// TIA Portal V20 export
FUNCTION_BLOCK "LER_E5CC"   // FB23, LAD
// stored: Access Published, MemoryReserve 100, SetENOAutomatically false
   VAR_INPUT
      enable : Bool;
      clock : Bool;
      unitNo : Int;
      save : Bool;
      Reset : Bool;
      AllHeaterRun : Bool;
      AllHeaterStop : Bool;
      AllHeaterAutoTuneRun : Bool;
      AllHeaterAutoTuneStop : Bool;
      HeaterCommands : "LER_typeE5CCCommands";
      HeaterConfiguration : "LER_typeE5CCConfiguration";
   END_VAR
   VAR_OUTPUT
      HeaterMonitoring : "LER_typeE5CCMonitoring";
   END_VAR
   VAR_IN_OUT
      CurrentUnit : Int;
      MBMasterBuffer : "LER_typeHeaterConfiguration_MB_Master";
   END_VAR
   VAR
      statHeaterRun : Bool;
      statHeaterStop : Bool;
      statHeaterAutoTuneRun : Bool;
      statHeaterAutoTuneStop : Bool;
      statReadStep : Int;
      statReadReq : Array[0..9] of Bool;
      statWriteReq : Array[0..9] of Bool;
      statPulse : Array[0..19] of Bool;
      statTimer { S7_SetPoint := 'True'} : Array[0..9] of TON_TIME;
      statReadTempPV : Real;
      statReadStatus : DWord;
      statTempSP : Real;
      statAlarmValue1 : Real;
      statAlarmValue1_UpperLimit : Real;
      statAlarmValue1_LowerLimit : Real;
      statAlarmValue2 : Real;
      statAlarmValue2_UpperLimit : Real;
      statAlarmValue2_LowerLimit : Real;
      statReadStatus_Bool : Array[0..31] of Bool;
      statHeater_PV_Buf : Real;
      statUpperComplete_Temp : Real;
      statLowerComplete_Temp : Real;
   END_VAR
   VAR_TEMP
      tempErr : Word;
   END_VAR
   VAR CONSTANT
      Addr_TempPV : UDInt := 40001;
      Addr_Status : UDInt := 40003;
      Addr_TempSP : UDInt := 40263;
      Addr_AlarmValue1 : UDInt := 40265;
      Addr_AlarmValue1_UpperLimit : UDInt := 40267;
      Addr_AlarmValue1_LowerLimit : UDInt := 40269;
      Addr_AlarmValue2 : UDInt := 40271;
      Addr_AlarmValue2_UpperLimit : UDInt := 40273;
      Addr_AlarmValue2_LowerLimit : UDInt := 40275;
      CMD_Run : DWord := 16#01000000;
      CMD_Stop : DWord := 16#01010000;
      CMD_AutoTune_Run : DWord := 16#03020000;
      CMD_AutoTune_Stop : DWord := 16#03000000;
      Mode_Read : Int := 0;
      Mode_Write : Int := 1;
      Read_Time : Time := T#1000MS;
      STATUS_NO_ERROR_OCCURRED : DWord;   // No error occurred.
      ERR_HEATER_CURRENT_VALUE_EXCEEDED_CT1 : DWord := 16#1;
      ERR_HEATER_CURRENT_VALUE_HOLD_CT1 : DWord := 16#2;
      ERR_AD_CONVERTER_ABNORMALITY : DWord := 16#4;
      ERR_HS_SSR_FAULT_ALERT_CT1 : DWord := 16#8;
      ERR_RSP_INPUT_ABNORMALITIES : DWord := 16#10;
      ERR_MORE_THAN_INPUT : DWord := 16#40;
      ERR_POTENTIOMETER_INPUT_ABNORMAL : DWord := 16#80;
      ERR_CONTROL_OUTPUT_HEATED_OPEN_OUTPUT : DWord := 16#100;
      ERR_CONTROL_OUTPUT_COOL_CLOSE_OUTPUT : DWord := 16#200;
      ERR_HEATER_OPEN_CIRCUIT_HB_ALARM_CT1 : DWord := 16#400;
      ERR_HEATER_OPEN_CIRCUIT_HB_ALARM_CT2 : DWord := 16#800;
      ERR_ALERT_1 : DWord := 16#1000;
      ERR_ALERT_2 : DWord := 16#2000;
      ERR_ALERT_3 : DWord := 16#4000;
      ERR_PROGRAM_END_OUTPUT : DWord := 16#8000;
      ERR_EVENT_INPUT_1 : DWord := 16#10000;
      ERR_EVENT_INPUT_2 : DWord := 16#20000;
      ERR_EVENT_INPUT_3 : DWord := 16#40000;
      ERR_EVENT_INPUT_4 : DWord := 16#80000;
      ERR_WRITE_MODE : DWord := 16#100000;
      ERR_NON_VOLATILE_MEMORY : DWord := 16#200000;
      ERR_SETTING_AREA : DWord := 16#400000;
      ERR_AT_RUN_STOP : DWord := 16#800000;
      ERR_RUN_STOP : DWord := 16#1000000;
      ERR_COMMUNICATION_WRITE : DWord := 16#2000000;
      ERR_AUTO_MANUAL : DWord := 16#4000000;
      ERR_PROGRAM_START : DWord := 16#8000000;
      ERR_HEATER_CURRENT_VALUE_EXCEEDED_CT2 : DWord := 16#10000000;
      ERR_HEATER_CURRENT_VALUE_HOLD_CT2 : DWord := 16#20000000;
      ERR_HS_SSR_FAILURE_ALARM_CT2 : DWord := 16#80000000;
   END_VAR
   // // statReadStatus_Bool[0] : Heater Current Value Exceeded (CT1)
   // // statReadStatus_Bool[1] : Heater Current Value Hold (CT1)
   // // statReadStatus_Bool[2] : AD converter abnormality
   // // statReadStatus_Bool[3] : HS (SSR Fault) Alert (CT1)
   // // statReadStatus_Bool[4] : RSP input abnormalities
   // // statReadStatus_Bool[6] : More than input
   // // statReadStatus_Bool[7] : Potenshometer input abnormal
   // // statReadStatus_Bool[8] : Control Output (Heated)/Open Output
   // // statReadStatus_Bool[9] : Control Output (Cool)/Close Output
   // // statReadStatus_Bool[10] : Heater Open Circuit (HB) Alarm (CT1)
   // // statReadStatus_Bool[11] : Heater Open Circuit (HB) Alarm (CT2)
   // // statReadStatus_Bool[12] : Alert 1
   // // statReadStatus_Bool[13] : Alert 2
   // // statReadStatus_Bool[14] : Alert 3
   // // statReadStatus_Bool[15] : Program END Output
   // // statReadStatus_Bool[16] : Event Input 1
   // // statReadStatus_Bool[17] : Event Input 2
   // // statReadStatus_Bool[18] : Event Input 3
   // // statReadStatus_Bool[19] : Event Input 4
   // // statReadStatus_Bool[20] : Write Mode
   // // statReadStatus_Bool[21] : Non-volatile Memory
   // // statReadStatus_Bool[22] : Setting Area
   // // statReadStatus_Bool[23] : AT Run/Stop
   // // statReadStatus_Bool[24] : RUN/STOP
   // // statReadStatus_Bool[25] : Communication Write
   // // statReadStatus_Bool[26] : Auto/Manual
   // // statReadStatus_Bool[27] : Program START
   // // statReadStatus_Bool[28] : Heater Current Value Exceeded (CT2)
   // // statReadStatus_Bool[29] : Heater Current Value Hold (CT2)
   // // statReadStatus_Bool[31] : HS (SSR Failure) Alarm (CT2)
   VAR_TEMP   // added for the SCL form of the ladder/FBD networks
      _w1 : Bool;
      _w2 : Bool;
   END_VAR
BEGIN

REGION Network 1 (SCL): ###### Input Mapping ######
   //Input Mapping
   #statHeaterRun := #AllHeaterRun OR #HeaterCommands.Heater_Run;
   #statHeaterStop := #AllHeaterStop OR #HeaterCommands.Heater_Stop;
   #statHeaterAutoTuneRun := #AllHeaterAutoTuneRun OR #HeaterCommands.AutoTune_Run;
   #statHeaterAutoTuneStop := #AllHeaterAutoTuneStop OR #HeaterCommands.AutoTune_Stop;

   //Read Step Initialization
   IF #statReadStep = 0 THEN
       #statReadStep := 1;
   ELSIF #statReadStep > 2 THEN
       #statReadStep := 1;
   END_IF;
END_REGION

REGION Network 2: Read Temp PV + Status Command
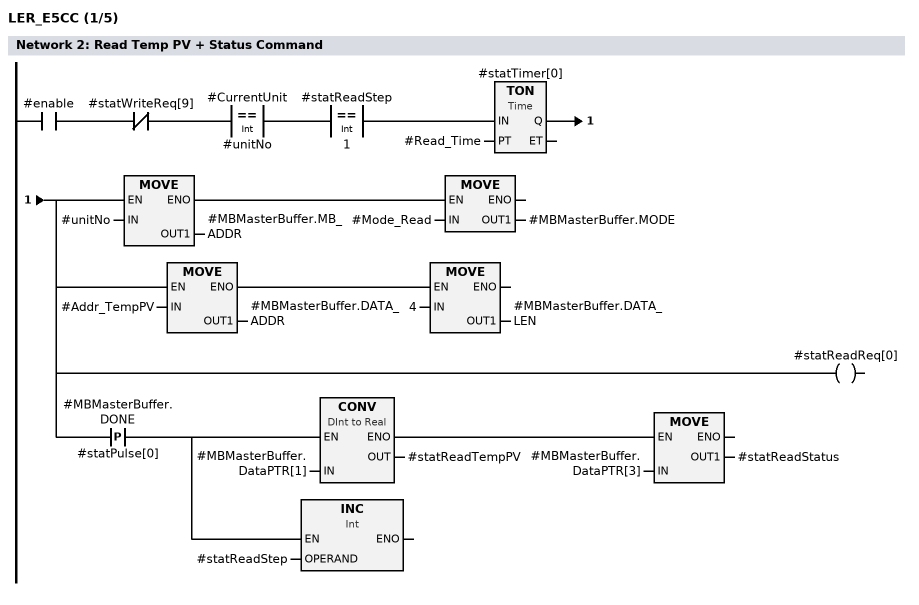
   RUNG wire#powerrail
      Contact( #enable )
      I_Contact( #statWriteReq[9] )
      { S7_Templates := "SrcType := Int" } EQ_Contact(in1 := #CurrentUnit, in2 := #unitNo)
      { S7_Templates := "SrcType := Int" } EQ_Contact(in1 := #statReadStep, in2 := 1)
      { S7_Templates := "time_type := Time" } #statTimer[0].TON(pt := #Read_Time, et =>)
      wire#w1
      Move(in := #unitNo, out1 => #MBMasterBuffer.MB_ADDR)
      Move(in := #Mode_Read, out1 => #MBMasterBuffer.MODE)
   END_RUNG
   RUNG wire#w1
      Move(in := #Addr_TempPV, out1 => #MBMasterBuffer.DATA_ADDR)
      Move(in := 4, out1 => #MBMasterBuffer.DATA_LEN)
   END_RUNG
   RUNG wire#w1
      Coil( #statReadReq[0] )
   END_RUNG
   RUNG wire#w1
      P_Contact(operand := #MBMasterBuffer.DONE, bit := #statPulse[0])
      wire#w2
      { S7_Templates := "[SrcType := DInt, DestType := Real]" } Convert(in := #MBMasterBuffer.DataPTR[1], out => #statReadTempPV)
      Move(in := #MBMasterBuffer.DataPTR[3], out1 => #statReadStatus)
   END_RUNG
   RUNG wire#w2
      { S7_Templates := "DestType := Int" } Inc( #statReadStep )
   END_RUNG
   // the same network as SCL:
   #statTimer[0].TON(IN := #enable AND NOT #statWriteReq[9] AND (#CurrentUnit = #unitNo) AND (#statReadStep = 1),
                     PT := #Read_Time);
   IF #statTimer[0].Q THEN
       #MBMasterBuffer.MB_ADDR := #unitNo;
       #MBMasterBuffer.MODE := #Mode_Read;
       #MBMasterBuffer.DATA_ADDR := #Addr_TempPV;
       #MBMasterBuffer.DATA_LEN := 4;
   END_IF;
   #statReadReq[0] := #statTimer[0].Q;
   #_w1 := #statTimer[0].Q AND #MBMasterBuffer.DONE AND NOT #statPulse[0];   // rising edge of #MBMasterBuffer.DONE
   #statPulse[0] := #MBMasterBuffer.DONE;
   IF #_w1 THEN
       #statReadTempPV := DINT_TO_REAL(#MBMasterBuffer.DataPTR[1]);
       #statReadStatus := #MBMasterBuffer.DataPTR[3];
       #statReadStep := #statReadStep + 1;
   END_IF;
END_REGION

REGION Network 3: Read TempSP + AlarmValue1 ~ AlarmValue2_LowerLimit Commad
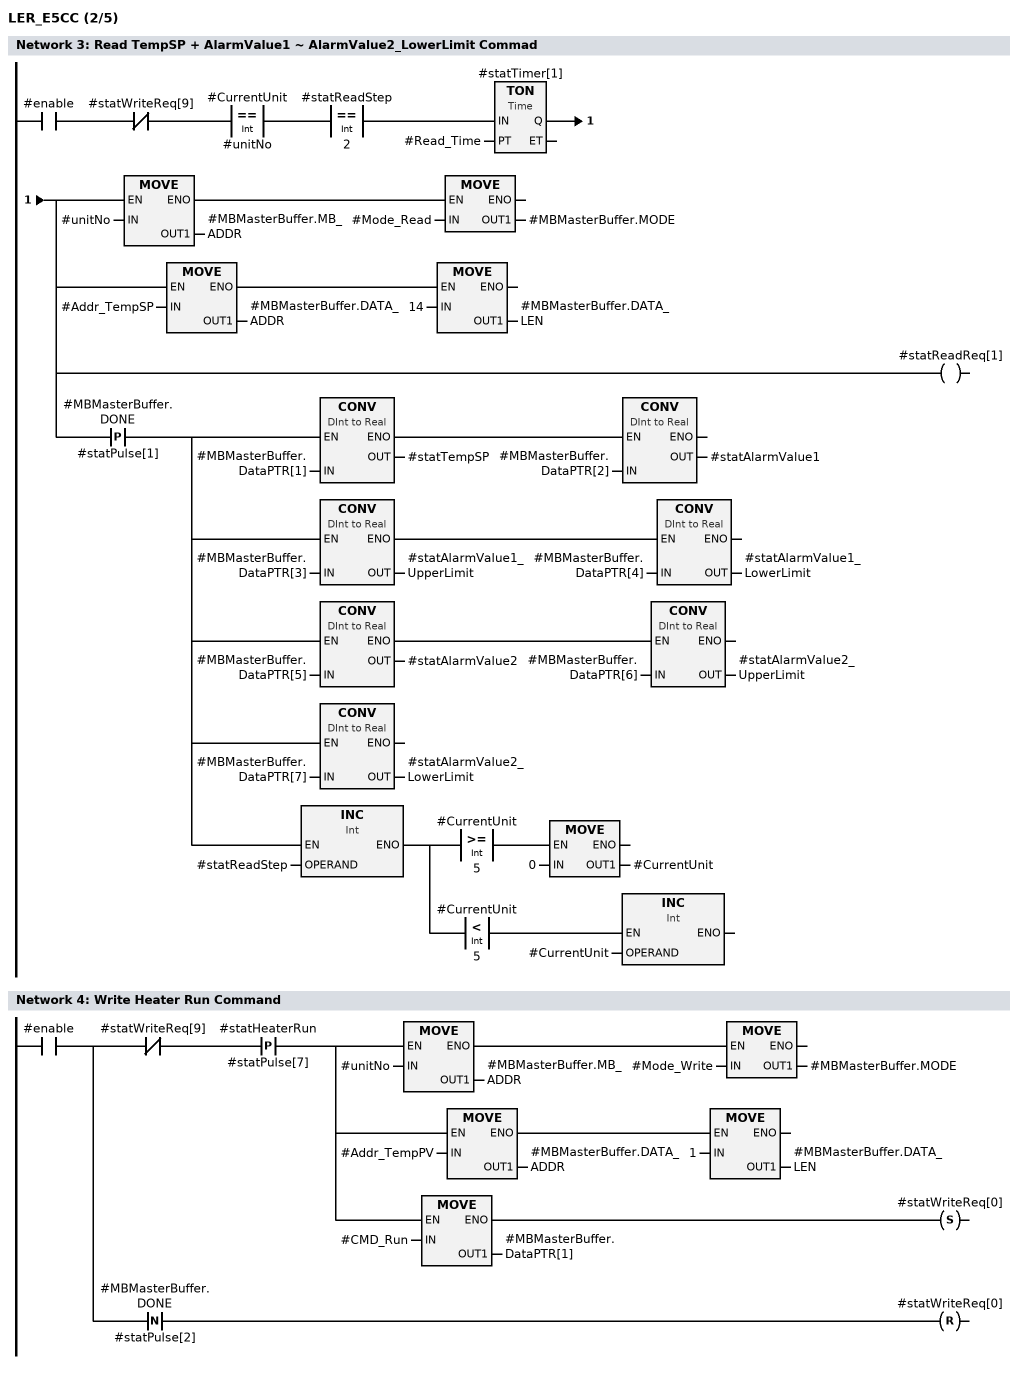
   RUNG wire#powerrail
      Contact( #enable )
      I_Contact( #statWriteReq[9] )
      { S7_Templates := "SrcType := Int" } EQ_Contact(in1 := #CurrentUnit, in2 := #unitNo)
      { S7_Templates := "SrcType := Int" } EQ_Contact(in1 := #statReadStep, in2 := 2)
      { S7_Templates := "time_type := Time" } #statTimer[1].TON(pt := #Read_Time, et =>)
      wire#w1
      Move(in := #unitNo, out1 => #MBMasterBuffer.MB_ADDR)
      Move(in := #Mode_Read, out1 => #MBMasterBuffer.MODE)
   END_RUNG
   RUNG wire#w1
      Move(in := #Addr_TempSP, out1 => #MBMasterBuffer.DATA_ADDR)
      Move(in := 14, out1 => #MBMasterBuffer.DATA_LEN)
   END_RUNG
   RUNG wire#w1
      Coil( #statReadReq[1] )
   END_RUNG
   RUNG wire#w1
      P_Contact(operand := #MBMasterBuffer.DONE, bit := #statPulse[1])
      wire#w2
      { S7_Templates := "[SrcType := DInt, DestType := Real]" } Convert(in := #MBMasterBuffer.DataPTR[1], out => #statTempSP)
      { S7_Templates := "[SrcType := DInt, DestType := Real]" } Convert(in := #MBMasterBuffer.DataPTR[2], out => #statAlarmValue1)
   END_RUNG
   RUNG wire#w2
      { S7_Templates := "[SrcType := DInt, DestType := Real]" } Convert(in := #MBMasterBuffer.DataPTR[3], out => #statAlarmValue1_UpperLimit)
      { S7_Templates := "[SrcType := DInt, DestType := Real]" } Convert(in := #MBMasterBuffer.DataPTR[4], out => #statAlarmValue1_LowerLimit)
   END_RUNG
   RUNG wire#w2
      { S7_Templates := "[SrcType := DInt, DestType := Real]" } Convert(in := #MBMasterBuffer.DataPTR[5], out => #statAlarmValue2)
      { S7_Templates := "[SrcType := DInt, DestType := Real]" } Convert(in := #MBMasterBuffer.DataPTR[6], out => #statAlarmValue2_UpperLimit)
   END_RUNG
   RUNG wire#w2
      { S7_Templates := "[SrcType := DInt, DestType := Real]" } Convert(in := #MBMasterBuffer.DataPTR[7], out => #statAlarmValue2_LowerLimit)
   END_RUNG
   RUNG wire#w2
      { S7_Templates := "DestType := Int" } Inc( #statReadStep )
      wire#w3
      { S7_Templates := "SrcType := Int" } GE_Contact(in1 := #CurrentUnit, in2 := 5)
      Move(in := 0, out1 => #CurrentUnit)
   END_RUNG
   RUNG wire#w3
      { S7_Templates := "SrcType := Int" } LT_Contact(in1 := #CurrentUnit, in2 := 5)
      { S7_Templates := "DestType := Int" } Inc( #CurrentUnit )
   END_RUNG
   // the same network as SCL:
   #statTimer[1].TON(IN := #enable AND NOT #statWriteReq[9] AND (#CurrentUnit = #unitNo) AND (#statReadStep = 2),
                     PT := #Read_Time);
   IF #statTimer[1].Q THEN
       #MBMasterBuffer.MB_ADDR := #unitNo;
       #MBMasterBuffer.MODE := #Mode_Read;
       #MBMasterBuffer.DATA_ADDR := #Addr_TempSP;
       #MBMasterBuffer.DATA_LEN := 14;
   END_IF;
   #statReadReq[1] := #statTimer[1].Q;
   #_w1 := #statTimer[1].Q AND #MBMasterBuffer.DONE AND NOT #statPulse[1];   // rising edge of #MBMasterBuffer.DONE
   #statPulse[1] := #MBMasterBuffer.DONE;
   IF #_w1 THEN
       #statTempSP := DINT_TO_REAL(#MBMasterBuffer.DataPTR[1]);
       #statAlarmValue1 := DINT_TO_REAL(#MBMasterBuffer.DataPTR[2]);
       #statAlarmValue1_UpperLimit := DINT_TO_REAL(#MBMasterBuffer.DataPTR[3]);
       #statAlarmValue1_LowerLimit := DINT_TO_REAL(#MBMasterBuffer.DataPTR[4]);
       #statAlarmValue2 := DINT_TO_REAL(#MBMasterBuffer.DataPTR[5]);
       #statAlarmValue2_UpperLimit := DINT_TO_REAL(#MBMasterBuffer.DataPTR[6]);
       #statAlarmValue2_LowerLimit := DINT_TO_REAL(#MBMasterBuffer.DataPTR[7]);
       #statReadStep := #statReadStep + 1;
   END_IF;
   IF #_w1 AND (#CurrentUnit >= 5) THEN #CurrentUnit := 0; END_IF;
   IF #_w1 AND (#CurrentUnit < 5) THEN #CurrentUnit := #CurrentUnit + 1; END_IF;
END_REGION

REGION Network 4: Write Heater Run Command
   RUNG wire#powerrail
      Contact( #enable )
      wire#w1
      I_Contact( #statWriteReq[9] )
      P_Contact(operand := #statHeaterRun, bit := #statPulse[7])
      wire#w2
      Move(in := #unitNo, out1 => #MBMasterBuffer.MB_ADDR)
      Move(in := #Mode_Write, out1 => #MBMasterBuffer.MODE)
   END_RUNG
   RUNG wire#w2
      Move(in := #Addr_TempPV, out1 => #MBMasterBuffer.DATA_ADDR)
      Move(in := 1, out1 => #MBMasterBuffer.DATA_LEN)
   END_RUNG
   RUNG wire#w2
      Move(in := #CMD_Run, out1 => #MBMasterBuffer.DataPTR[1])
      S_Coil( #statWriteReq[0] )
   END_RUNG
   RUNG wire#w1
      N_Contact(operand := #MBMasterBuffer.DONE, bit := #statPulse[2])
      R_Coil( #statWriteReq[0] )
   END_RUNG
   // the same network as SCL:
   #_w1 := #enable AND NOT #statWriteReq[9] AND #statHeaterRun AND NOT #statPulse[7];   // rising edge of #statHeaterRun
   #statPulse[7] := #statHeaterRun;
   IF #_w1 THEN
       #MBMasterBuffer.MB_ADDR := #unitNo;
       #MBMasterBuffer.MODE := #Mode_Write;
       #MBMasterBuffer.DATA_ADDR := #Addr_TempPV;
       #MBMasterBuffer.DATA_LEN := 1;
       #MBMasterBuffer.DataPTR[1] := #CMD_Run;
       #statWriteReq[0] := TRUE;
   END_IF;
   #_w2 := #enable AND NOT #MBMasterBuffer.DONE AND #statPulse[2];   // falling edge of #MBMasterBuffer.DONE
   #statPulse[2] := #MBMasterBuffer.DONE;
   IF #_w2 THEN #statWriteReq[0] := FALSE; END_IF;
END_REGION

REGION Network 5: Write Heater Stop Command
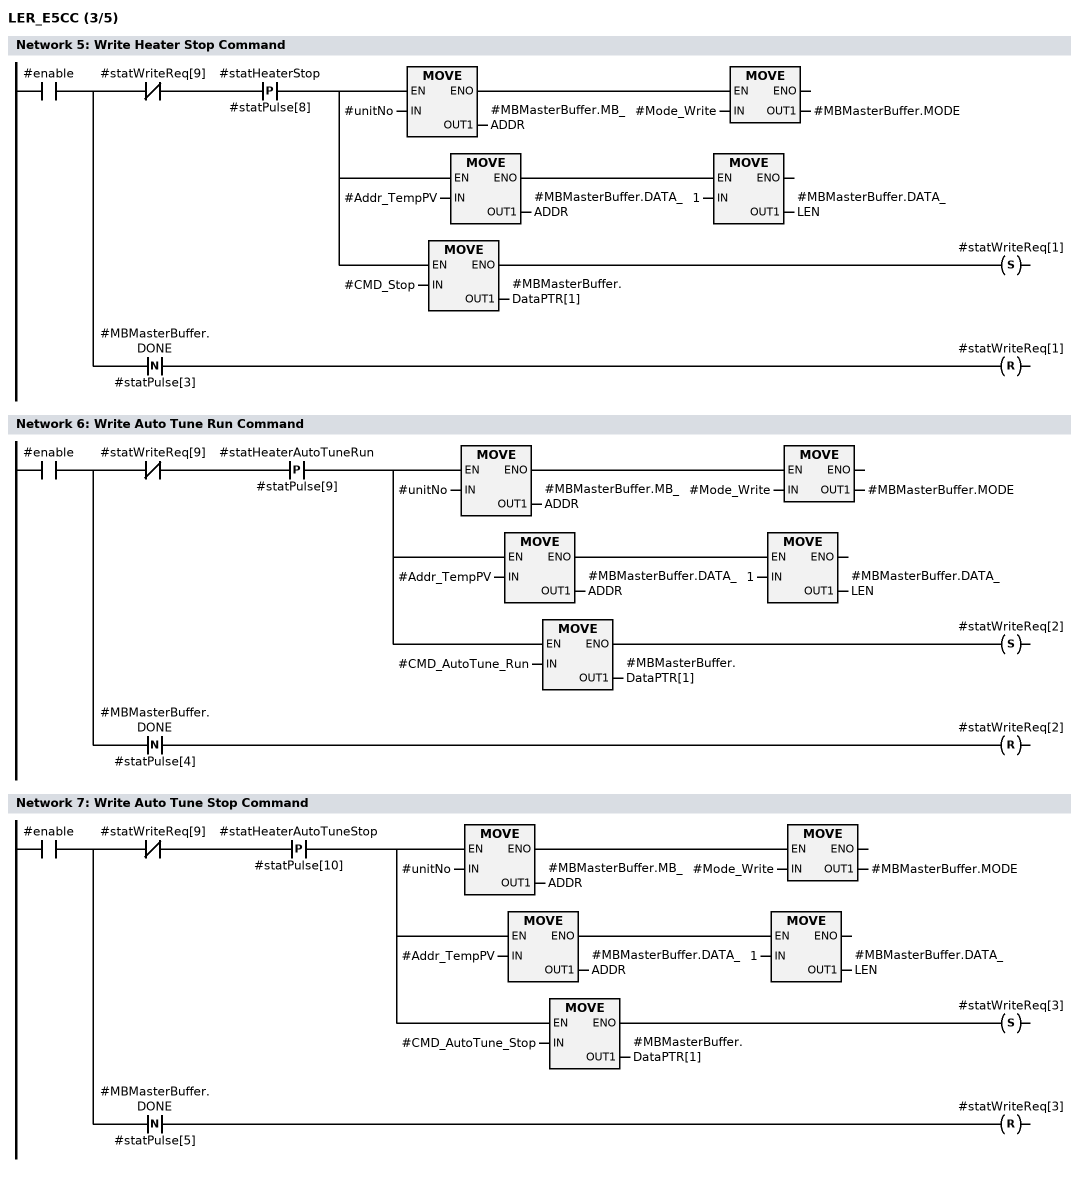
   RUNG wire#powerrail
      Contact( #enable )
      wire#w1
      I_Contact( #statWriteReq[9] )
      P_Contact(operand := #statHeaterStop, bit := #statPulse[8])
      wire#w2
      Move(in := #unitNo, out1 => #MBMasterBuffer.MB_ADDR)
      Move(in := #Mode_Write, out1 => #MBMasterBuffer.MODE)
   END_RUNG
   RUNG wire#w2
      Move(in := #Addr_TempPV, out1 => #MBMasterBuffer.DATA_ADDR)
      Move(in := 1, out1 => #MBMasterBuffer.DATA_LEN)
   END_RUNG
   RUNG wire#w2
      Move(in := #CMD_Stop, out1 => #MBMasterBuffer.DataPTR[1])
      S_Coil( #statWriteReq[1] )
   END_RUNG
   RUNG wire#w1
      N_Contact(operand := #MBMasterBuffer.DONE, bit := #statPulse[3])
      R_Coil( #statWriteReq[1] )
   END_RUNG
   // the same network as SCL:
   #_w1 := #enable AND NOT #statWriteReq[9] AND #statHeaterStop AND NOT #statPulse[8];   // rising edge of #statHeaterStop
   #statPulse[8] := #statHeaterStop;
   IF #_w1 THEN
       #MBMasterBuffer.MB_ADDR := #unitNo;
       #MBMasterBuffer.MODE := #Mode_Write;
       #MBMasterBuffer.DATA_ADDR := #Addr_TempPV;
       #MBMasterBuffer.DATA_LEN := 1;
       #MBMasterBuffer.DataPTR[1] := #CMD_Stop;
       #statWriteReq[1] := TRUE;
   END_IF;
   #_w2 := #enable AND NOT #MBMasterBuffer.DONE AND #statPulse[3];   // falling edge of #MBMasterBuffer.DONE
   #statPulse[3] := #MBMasterBuffer.DONE;
   IF #_w2 THEN #statWriteReq[1] := FALSE; END_IF;
END_REGION

REGION Network 6: Write Auto Tune Run Command
   RUNG wire#powerrail
      Contact( #enable )
      wire#w1
      I_Contact( #statWriteReq[9] )
      P_Contact(operand := #statHeaterAutoTuneRun, bit := #statPulse[9])
      wire#w2
      Move(in := #unitNo, out1 => #MBMasterBuffer.MB_ADDR)
      Move(in := #Mode_Write, out1 => #MBMasterBuffer.MODE)
   END_RUNG
   RUNG wire#w2
      Move(in := #Addr_TempPV, out1 => #MBMasterBuffer.DATA_ADDR)
      Move(in := 1, out1 => #MBMasterBuffer.DATA_LEN)
   END_RUNG
   RUNG wire#w2
      Move(in := #CMD_AutoTune_Run, out1 => #MBMasterBuffer.DataPTR[1])
      S_Coil( #statWriteReq[2] )
   END_RUNG
   RUNG wire#w1
      N_Contact(operand := #MBMasterBuffer.DONE, bit := #statPulse[4])
      R_Coil( #statWriteReq[2] )
   END_RUNG
   // the same network as SCL:
   #_w1 := #enable AND NOT #statWriteReq[9] AND #statHeaterAutoTuneRun AND NOT #statPulse[9];   // rising edge of #statHeaterAutoTuneRun
   #statPulse[9] := #statHeaterAutoTuneRun;
   IF #_w1 THEN
       #MBMasterBuffer.MB_ADDR := #unitNo;
       #MBMasterBuffer.MODE := #Mode_Write;
       #MBMasterBuffer.DATA_ADDR := #Addr_TempPV;
       #MBMasterBuffer.DATA_LEN := 1;
       #MBMasterBuffer.DataPTR[1] := #CMD_AutoTune_Run;
       #statWriteReq[2] := TRUE;
   END_IF;
   #_w2 := #enable AND NOT #MBMasterBuffer.DONE AND #statPulse[4];   // falling edge of #MBMasterBuffer.DONE
   #statPulse[4] := #MBMasterBuffer.DONE;
   IF #_w2 THEN #statWriteReq[2] := FALSE; END_IF;
END_REGION

REGION Network 7: Write Auto Tune Stop Command
   RUNG wire#powerrail
      Contact( #enable )
      wire#w1
      I_Contact( #statWriteReq[9] )
      P_Contact(operand := #statHeaterAutoTuneStop, bit := #statPulse[10])
      wire#w2
      Move(in := #unitNo, out1 => #MBMasterBuffer.MB_ADDR)
      Move(in := #Mode_Write, out1 => #MBMasterBuffer.MODE)
   END_RUNG
   RUNG wire#w2
      Move(in := #Addr_TempPV, out1 => #MBMasterBuffer.DATA_ADDR)
      Move(in := 1, out1 => #MBMasterBuffer.DATA_LEN)
   END_RUNG
   RUNG wire#w2
      Move(in := #CMD_AutoTune_Stop, out1 => #MBMasterBuffer.DataPTR[1])
      S_Coil( #statWriteReq[3] )
   END_RUNG
   RUNG wire#w1
      N_Contact(operand := #MBMasterBuffer.DONE, bit := #statPulse[5])
      R_Coil( #statWriteReq[3] )
   END_RUNG
   // the same network as SCL:
   #_w1 := #enable AND NOT #statWriteReq[9] AND #statHeaterAutoTuneStop AND NOT #statPulse[10];   // rising edge of #statHeaterAutoTuneStop
   #statPulse[10] := #statHeaterAutoTuneStop;
   IF #_w1 THEN
       #MBMasterBuffer.MB_ADDR := #unitNo;
       #MBMasterBuffer.MODE := #Mode_Write;
       #MBMasterBuffer.DATA_ADDR := #Addr_TempPV;
       #MBMasterBuffer.DATA_LEN := 1;
       #MBMasterBuffer.DataPTR[1] := #CMD_AutoTune_Stop;
       #statWriteReq[3] := TRUE;
   END_IF;
   #_w2 := #enable AND NOT #MBMasterBuffer.DONE AND #statPulse[5];   // falling edge of #MBMasterBuffer.DONE
   #statPulse[5] := #MBMasterBuffer.DONE;
   IF #_w2 THEN #statWriteReq[3] := FALSE; END_IF;
END_REGION

REGION Network 8: Write TempSP + AlarmValue1 ~ AlarmValue2_LowerLimit Command
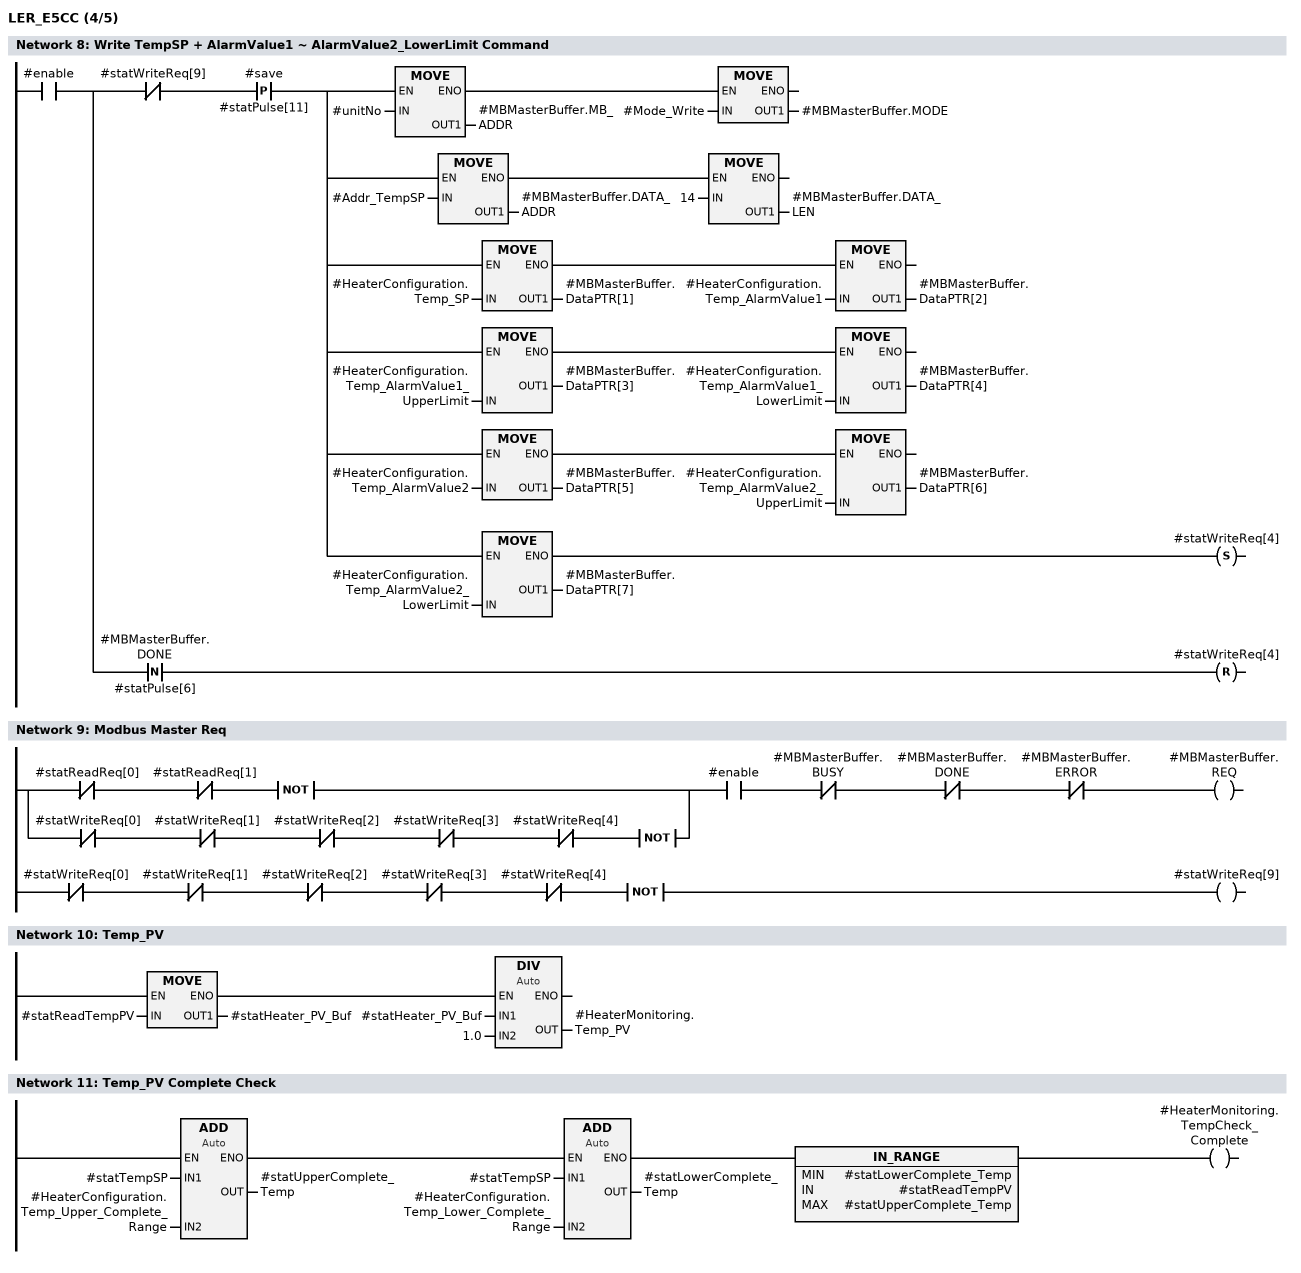
   RUNG wire#powerrail
      Contact( #enable )
      wire#w1
      I_Contact( #statWriteReq[9] )
      P_Contact(operand := #save, bit := #statPulse[11])
      wire#w2
      Move(in := #unitNo, out1 => #MBMasterBuffer.MB_ADDR)
      Move(in := #Mode_Write, out1 => #MBMasterBuffer.MODE)
   END_RUNG
   RUNG wire#w2
      Move(in := #Addr_TempSP, out1 => #MBMasterBuffer.DATA_ADDR)
      Move(in := 14, out1 => #MBMasterBuffer.DATA_LEN)
   END_RUNG
   RUNG wire#w2
      Move(in := #HeaterConfiguration.Temp_SP, out1 => #MBMasterBuffer.DataPTR[1])
      Move(in := #HeaterConfiguration.Temp_AlarmValue1, out1 => #MBMasterBuffer.DataPTR[2])
   END_RUNG
   RUNG wire#w2
      Move(in := #HeaterConfiguration.Temp_AlarmValue1_UpperLimit, out1 => #MBMasterBuffer.DataPTR[3])
      Move(in := #HeaterConfiguration.Temp_AlarmValue1_LowerLimit, out1 => #MBMasterBuffer.DataPTR[4])
   END_RUNG
   RUNG wire#w2
      Move(in := #HeaterConfiguration.Temp_AlarmValue2, out1 => #MBMasterBuffer.DataPTR[5])
      Move(in := #HeaterConfiguration.Temp_AlarmValue2_UpperLimit, out1 => #MBMasterBuffer.DataPTR[6])
   END_RUNG
   RUNG wire#w2
      Move(in := #HeaterConfiguration.Temp_AlarmValue2_LowerLimit, out1 => #MBMasterBuffer.DataPTR[7])
      S_Coil( #statWriteReq[4] )
   END_RUNG
   RUNG wire#w1
      N_Contact(operand := #MBMasterBuffer.DONE, bit := #statPulse[6])
      R_Coil( #statWriteReq[4] )
   END_RUNG
   // the same network as SCL:
   #_w1 := #enable AND NOT #statWriteReq[9] AND #save AND NOT #statPulse[11];   // rising edge of #save
   #statPulse[11] := #save;
   IF #_w1 THEN
       #MBMasterBuffer.MB_ADDR := #unitNo;
       #MBMasterBuffer.MODE := #Mode_Write;
       #MBMasterBuffer.DATA_ADDR := #Addr_TempSP;
       #MBMasterBuffer.DATA_LEN := 14;
       #MBMasterBuffer.DataPTR[1] := #HeaterConfiguration.Temp_SP;
       #MBMasterBuffer.DataPTR[2] := #HeaterConfiguration.Temp_AlarmValue1;
       #MBMasterBuffer.DataPTR[3] := #HeaterConfiguration.Temp_AlarmValue1_UpperLimit;
       #MBMasterBuffer.DataPTR[4] := #HeaterConfiguration.Temp_AlarmValue1_LowerLimit;
       #MBMasterBuffer.DataPTR[5] := #HeaterConfiguration.Temp_AlarmValue2;
       #MBMasterBuffer.DataPTR[6] := #HeaterConfiguration.Temp_AlarmValue2_UpperLimit;
       #MBMasterBuffer.DataPTR[7] := #HeaterConfiguration.Temp_AlarmValue2_LowerLimit;
       #statWriteReq[4] := TRUE;
   END_IF;
   #_w2 := #enable AND NOT #MBMasterBuffer.DONE AND #statPulse[6];   // falling edge of #MBMasterBuffer.DONE
   #statPulse[6] := #MBMasterBuffer.DONE;
   IF #_w2 THEN #statWriteReq[4] := FALSE; END_IF;
END_REGION

REGION Network 9: Modbus Master Req
   RUNG wire#powerrail
      I_Contact( #statReadReq[0] )
      I_Contact( #statReadReq[1] )
      Not()
      wire#w1
      Contact( #enable )
      I_Contact( #MBMasterBuffer.BUSY )
      I_Contact( #MBMasterBuffer.DONE )
      I_Contact( #MBMasterBuffer.ERROR )
      Coil( #MBMasterBuffer.REQ )
   END_RUNG
   RUNG wire#powerrail
      I_Contact( #statWriteReq[0] )
      I_Contact( #statWriteReq[1] )
      I_Contact( #statWriteReq[2] )
      I_Contact( #statWriteReq[3] )
      I_Contact( #statWriteReq[4] )
      Not()
   END_RUNG wire#w1
   RUNG wire#powerrail
      I_Contact( #statWriteReq[0] )
      I_Contact( #statWriteReq[1] )
      I_Contact( #statWriteReq[2] )
      I_Contact( #statWriteReq[3] )
      I_Contact( #statWriteReq[4] )
      Not()
      Coil( #statWriteReq[9] )
   END_RUNG
   // the same network as SCL:
   #MBMasterBuffer.REQ := (NOT (NOT #statReadReq[0] AND NOT #statReadReq[1]) OR NOT (NOT #statWriteReq[0] AND NOT #statWriteReq[1] AND NOT #statWriteReq[2] AND NOT #statWriteReq[3] AND NOT #statWriteReq[4])) AND #enable AND NOT #MBMasterBuffer.BUSY AND NOT #MBMasterBuffer.DONE AND NOT #MBMasterBuffer.ERROR;
   #statWriteReq[9] := NOT (NOT #statWriteReq[0] AND NOT #statWriteReq[1] AND NOT #statWriteReq[2] AND NOT #statWriteReq[3] AND NOT #statWriteReq[4]);
END_REGION

REGION Network 10: Temp_PV
   RUNG wire#powerrail
      Move(in := #statReadTempPV, out1 => #statHeater_PV_Buf)
      Div(in1 := #statHeater_PV_Buf, in2 := 1.0, out => #HeaterMonitoring.Temp_PV)
   END_RUNG
   // the same network as SCL:
   #statHeater_PV_Buf := #statReadTempPV;
   #HeaterMonitoring.Temp_PV := #statHeater_PV_Buf / 1.0;
END_REGION

REGION Network 11: Temp_PV Complete Check
   RUNG wire#powerrail
      Add(in1 := #statTempSP, in2 := #HeaterConfiguration.Temp_Upper_Complete_Range, out => #statUpperComplete_Temp)
      Add(in1 := #statTempSP, in2 := #HeaterConfiguration.Temp_Lower_Complete_Range, out => #statLowerComplete_Temp)
      { S7_Templates := "SrcType := Real" } InRange(min := #statLowerComplete_Temp, in := #statReadTempPV, max := #statUpperComplete_Temp)
      Coil( #HeaterMonitoring.TempCheck_Complete )
   END_RUNG
   // the same network as SCL:
   #statUpperComplete_Temp := #statTempSP + #HeaterConfiguration.Temp_Upper_Complete_Range;
   #statLowerComplete_Temp := #statTempSP + #HeaterConfiguration.Temp_Lower_Complete_Range;
   #HeaterMonitoring.TempCheck_Complete := (#statLowerComplete_Temp <= #statReadTempPV) AND (#statReadTempPV <= #statUpperComplete_Temp);
END_REGION

REGION Network 12: Heater Run Lamp
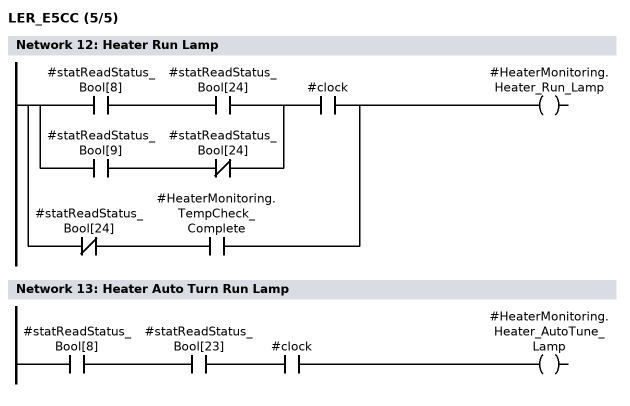
   RUNG wire#powerrail
      Contact( #statReadStatus_Bool[8] )
      Contact( #statReadStatus_Bool[24] )
      wire#w1
      Contact( #clock )
      wire#w2
      Coil( #HeaterMonitoring.Heater_Run_Lamp )
   END_RUNG
   RUNG wire#powerrail
      Contact( #statReadStatus_Bool[9] )
      I_Contact( #statReadStatus_Bool[24] )
   END_RUNG wire#w1
   RUNG wire#powerrail
      I_Contact( #statReadStatus_Bool[24] )
      Contact( #HeaterMonitoring.TempCheck_Complete )
   END_RUNG wire#w2
   // the same network as SCL:
   #HeaterMonitoring.Heater_Run_Lamp := (((#statReadStatus_Bool[8] AND #statReadStatus_Bool[24]) OR (#statReadStatus_Bool[9] AND NOT #statReadStatus_Bool[24])) AND #clock) OR (NOT #statReadStatus_Bool[24] AND #HeaterMonitoring.TempCheck_Complete);
END_REGION

REGION Network 13: Heater Auto Turn Run Lamp
   RUNG wire#powerrail
      Contact( #statReadStatus_Bool[8] )
      Contact( #statReadStatus_Bool[23] )
      Contact( #clock )
      Coil( #HeaterMonitoring.Heater_AutoTune_Lamp )
   END_RUNG
   // the same network as SCL:
   #HeaterMonitoring.Heater_AutoTune_Lamp := #statReadStatus_Bool[8] AND #statReadStatus_Bool[23] AND #clock;
END_REGION

REGION Network 14 (SCL): Error Check
   REGION  E5CC Error Status
       // Dword to Bool
       SCATTER(IN := #statReadStatus,
               OUT => #statReadStatus_Bool);
   END_REGION


   REGION Error Code Search
       IF #statReadStatus <> 0 THEN
           CASE #statReadStatus OF
               #ERR_HEATER_CURRENT_VALUE_EXCEEDED_CT1:
                   #HeaterMonitoring.Status := #ERR_HEATER_CURRENT_VALUE_EXCEEDED_CT1;
               #ERR_HEATER_CURRENT_VALUE_HOLD_CT1:
                   #HeaterMonitoring.Status := #ERR_HEATER_CURRENT_VALUE_HOLD_CT1;
               #ERR_AD_CONVERTER_ABNORMALITY:
                   #HeaterMonitoring.Status := #ERR_AD_CONVERTER_ABNORMALITY;
               #ERR_HS_SSR_FAULT_ALERT_CT1:
                   #HeaterMonitoring.Status := #ERR_HS_SSR_FAULT_ALERT_CT1;
               #ERR_RSP_INPUT_ABNORMALITIES:
                   #HeaterMonitoring.Status := #ERR_RSP_INPUT_ABNORMALITIES;
               #ERR_MORE_THAN_INPUT:
                   #HeaterMonitoring.Status := #ERR_MORE_THAN_INPUT;
               #ERR_POTENTIOMETER_INPUT_ABNORMAL:
                   #HeaterMonitoring.Status := #ERR_POTENTIOMETER_INPUT_ABNORMAL;
               #ERR_CONTROL_OUTPUT_HEATED_OPEN_OUTPUT:
                   #HeaterMonitoring.Status := #ERR_CONTROL_OUTPUT_HEATED_OPEN_OUTPUT;
               #ERR_CONTROL_OUTPUT_COOL_CLOSE_OUTPUT:
                   #HeaterMonitoring.Status := #ERR_CONTROL_OUTPUT_COOL_CLOSE_OUTPUT;
               #ERR_HEATER_OPEN_CIRCUIT_HB_ALARM_CT1:
                   #HeaterMonitoring.Status := #ERR_HEATER_OPEN_CIRCUIT_HB_ALARM_CT1;
               #ERR_HEATER_OPEN_CIRCUIT_HB_ALARM_CT2:
                   #HeaterMonitoring.Status := #ERR_HEATER_OPEN_CIRCUIT_HB_ALARM_CT2;
               #ERR_ALERT_1:
                   #HeaterMonitoring.Status := #ERR_ALERT_1;
               #ERR_ALERT_2:
                   #HeaterMonitoring.Status := #ERR_ALERT_2;
               #ERR_ALERT_3:
                   #HeaterMonitoring.Status := #ERR_ALERT_3;
               #ERR_PROGRAM_END_OUTPUT:
                   #HeaterMonitoring.Status := #ERR_PROGRAM_END_OUTPUT;
               #ERR_EVENT_INPUT_1:
                   #HeaterMonitoring.Status := #ERR_EVENT_INPUT_1;
               #ERR_EVENT_INPUT_2:
                   #HeaterMonitoring.Status := #ERR_EVENT_INPUT_2;
               #ERR_EVENT_INPUT_3:
                   #HeaterMonitoring.Status := #ERR_EVENT_INPUT_3;
               #ERR_EVENT_INPUT_4:
                   #HeaterMonitoring.Status := #ERR_EVENT_INPUT_4;
               #ERR_WRITE_MODE:
                   #HeaterMonitoring.Status := #ERR_WRITE_MODE;
               #ERR_NON_VOLATILE_MEMORY:
                   #HeaterMonitoring.Status := #ERR_NON_VOLATILE_MEMORY;
               #ERR_SETTING_AREA:
                   #HeaterMonitoring.Status := #ERR_SETTING_AREA;
               #ERR_AT_RUN_STOP:
                   #HeaterMonitoring.Status := #ERR_AT_RUN_STOP;
               #ERR_RUN_STOP:
                   #HeaterMonitoring.Status := #ERR_RUN_STOP;
               #ERR_COMMUNICATION_WRITE:
                   #HeaterMonitoring.Status := #ERR_COMMUNICATION_WRITE;
               #ERR_AUTO_MANUAL:
                   #HeaterMonitoring.Status := #ERR_AUTO_MANUAL;
               #ERR_PROGRAM_START:
                   #HeaterMonitoring.Status := #ERR_PROGRAM_START;
               #ERR_HEATER_CURRENT_VALUE_EXCEEDED_CT2:
                   #HeaterMonitoring.Status := #ERR_HEATER_CURRENT_VALUE_EXCEEDED_CT2;
               #ERR_HEATER_CURRENT_VALUE_HOLD_CT2:
                   #HeaterMonitoring.Status := #ERR_HEATER_CURRENT_VALUE_HOLD_CT2;
               #ERR_HS_SSR_FAILURE_ALARM_CT2:
                   #HeaterMonitoring.Status := #ERR_HS_SSR_FAILURE_ALARM_CT2;
           END_CASE;
       ELSIF #statReadStatus = 0 THEN
           #HeaterMonitoring.Status := 0;
       END_IF;
   END_REGION

   #HeaterMonitoring.Error := #statReadStatus <> 0;
END_REGION

REGION Network 15 (SCL): ##### Outputs mapping #####
   // Output Mapping
   #HeaterMonitoring.Temp_SP := #statTempSP;
   #HeaterMonitoring.Temp_AlarmValue1 := #statAlarmValue1;
   #HeaterMonitoring.Temp_AlarmValue1_UpperLimit := #statAlarmValue1_UpperLimit;
   #HeaterMonitoring.Temp_AlarmValue1_LowerLimit := #statAlarmValue1_LowerLimit;
   #HeaterMonitoring.Temp_AlarmValue2 := #statAlarmValue2;
   #HeaterMonitoring.Temp_AlarmValue2_UpperLimit := #statAlarmValue2_UpperLimit;
   #HeaterMonitoring.Temp_AlarmValue2_LowerLimit := #statAlarmValue2_LowerLimit;
   #HeaterMonitoring.E5CC_Status := #statReadStatus;
   #HeaterMonitoring.E5CC_Status_Bool := #statReadStatus_Bool;
END_REGION
END_FUNCTION_BLOCK
